// TwinCAT 3 PLC project PLC_project
// ProgramVersion: 3.1.4024.0
// libraries:
//   Tc2_Standard, * (Beckhoff Automation GmbH)
//   Tc2_System, * (Beckhoff Automation GmbH)
//   Tc3_Module, * (Beckhoff Automation GmbH)
// project tree:
//   Interface/ gOpc.TcGVL, TYP_BUTTONS_HW_IN.TcDUT, TYP_VESSEL_HW.TcDUT (not stored), TYP_VESSEL_HW_IN.TcDUT, TYP_VESSEL_HW_OUT.TcDUT (not stored)
//   / PlcTask.TcTTO
//   Main/ MAIN.TcPOU
// real-time tasks:
//   TASK PlcTask: cycle T#10ms, priority 20, ADS port 350

CONFIGURATION PLC_project
    RESOURCE PLC ON TwinCAT3
        TASK PlcTask(INTERVAL := T#10ms, PRIORITY := 20);
        PROGRAM MAIN WITH PlcTask : MAIN;
    END_RESOURCE
END_CONFIGURATION

// ---- Interface/TYP_BUTTONS_HW_IN.TcDUT
TYPE TYP_BUTTONS_HW_IN :
STRUCT
	ModeButton : BOOL; // false - state = MANUAL; true - state = AUTOMATIC
	AnalogButtons : ARRAY [1..2] OF REAL; // in manual mode button 1 = Max value for vessel 2 pressure; 2 = Min value for vessel 2 pressure
END_STRUCT
END_TYPE

// ---- Interface/TYP_VESSEL_HW_IN.TcDUT
TYPE TYP_VESSEL_HW_IN :
STRUCT
	Sensor : REAL; //pressure of the vessel
END_STRUCT
END_TYPE

// ---- Interface/gOpc.TcGVL
{attribute 'qualified_only'}
VAR_GLOBAL
	Vessel : ARRAY [1..2] OF TYP_VESSEL_HW;
	Buttons : TYP_BUTTONS_HW_IN;
	
END_VAR

// ---- Main/MAIN.TcPOU
PROGRAM MAIN
VAR
END_VAR

END_PROGRAM
